// TwinCAT 3 PLC project Untitled1
// ProgramVersion: 3.1.4023.0
// libraries:
//   Tc2_Standard, * (Beckhoff Automation GmbH)
//   Tc2_System, * (Beckhoff Automation GmbH)
//   Tc3_Module, * (Beckhoff Automation GmbH)
// project tree:
//   / ClassDiagram.TcCD (not stored), PlcTask.TcTTO (not stored)
//   Creator/ FB_ShapeCreator.TcPOU (not stored), FB_ShapeCreatorEX.TcPOU (not stored)
//   DUTs/ E_Shape.TcDUT (not stored)
//   Interfaces/ I_Shape.TcIO (not stored)
//   POUs/ MAIN.TcPOU
//   Shapes/ FB_Circle.TcPOU (not stored), FB_CustomShape.TcPOU (not stored), FB_Rectangle.TcPOU (not stored), FB_Square.TcPOU (not stored), FB_Star.TcPOU (not stored), FB_Triangle.TcPOU (not stored)
// real-time tasks:
//   TASK PlcTask: cycle T#10ms, priority 20, ADS port 350

// ---- POUs/MAIN.TcPOU
PROGRAM MAIN
VAR
	fbShapeCreator : FB_ShapeCreator;
//	fbShapeCreator : FB_ShapeCreatorEX;
	eShape : E_Shape := E_Shape.init;
	
	iShape : I_Shape;
END_VAR

fbShapeCreator(eShape:= eShape);

CASE eShape OF
	E_Shape.Circle:
		iShape := fbShapeCreator.M_GetShapeObject();
		IF iShape <> 0 THEN
			iShape.M_Draw();
		END_IF	
	
		eShape := E_Shape.Rectangle;
	
	E_Shape.Rectangle:
		iShape := fbShapeCreator.M_GetShapeObject();
		IF iShape <> 0 THEN
			iShape.M_Draw();
		END_IF
		
		eShape := E_Shape.Sqaure;	
		
	E_Shape.Sqaure:
		iShape := fbShapeCreator.M_GetShapeObject();
		IF iShape <> 0 THEN
			iShape.M_Draw();
		END_IF	
	
		eShape := E_Shape.Star;	

	E_Shape.Star:
		iShape := fbShapeCreator.M_GetShapeObject();
		IF iShape <> 0 THEN
			iShape.M_Draw();
		END_IF
		
		eShape := E_Shape.Triangle;	
	
	E_Shape.Triangle:
		iShape := fbShapeCreator.M_GetShapeObject();
		IF iShape <> 0 THEN
			iShape.M_Draw();
		END_IF	
	
		//eShape := E_Shape.end;	
		eShape := E_Shape.Custom;	
		
	E_Shape.Custom:
		iShape := fbShapeCreator.M_GetShapeObject();
		IF iShape <> 0 THEN
			iShape.M_Draw();
		END_IF
		
		eShape := E_Shape.end;	
END_CASE

END_PROGRAM
